      PresPreparada_M430 : Bool;
      PresMultiple_M430 : Bool;
      Bit_07_M430 : Bool;
      RecepOK_M431 : Bool;
      PresNormal_M431 : Bool;
      Ausencia_M431 : Bool;
      PresBloqueo_M431 : Bool;
      Galibo_M431 : Bool;
      PresPreparada_M431 : Bool;
      PresMultiple_M431 : Bool;
      Bit_07_M431 : Bool;
      RecepOK_M432 : Bool;
      PresNormal_M432 : Bool;
      Ausencia_M432 : Bool;
      PresBloqueo_M432 : Bool;
      Galibo_M432 : Bool;
      PresPreparada_M432 : Bool;
      PresMultiple_M432 : Bool;
      Bit_07_M432 : Bool;
      RecepOK_M433 : Bool;
      PresNormal_M433 : Bool;
      Ausencia_M433 : Bool;
      PresBloqueo_M433 : Bool;
      Galibo_M433 : Bool;
      PresPreparada_M433 : Bool;
      PresMultiple_M433 : Bool;
      Bit_07_M433 : Bool;
      RecepOK_M434 : Bool;
      PresNormal_M434 : Bool;
      Ausencia_M434 : Bool;
      PresBloqueo_M434 : Bool;
      Galibo_M434 : Bool;
      PresPreparada_M434 : Bool;
      PresMultiple_M434 : Bool;
      Bit_07_M434 : Bool;
      RecepOK_M435 : Bool;
      PresNormal_M435 : Bool;
      Ausencia_M435 : Bool;
      PresBloqueo_M435 : Bool;
      Galibo_M435 : Bool;
      PresPreparada_M435 : Bool;
      PresMultiple_M435 : Bool;
      Bit_07_M435 : Bool;
      RecepOK_M436 : Bool;
      PresNormal_M436 : Bool;
      Ausencia_M436 : Bool;
      PresBloqueo_M436 : Bool;
      Galibo_M436 : Bool;
      PresPreparada_M436 : Bool;
      PresMultiple_M436 : Bool;
      Bit_07_M436 : Bool;
      RecepOK_M437 : Bool;
      PresNormal_M437 : Bool;
      Ausencia_M437 : Bool;
      PresBloqueo_M437 : Bool;
      Galibo_M437 : Bool;
      PresPreparada_M437 : Bool;
      PresMultiple_M437 : Bool;
      Bit_07_M437 : Bool;
      RecepOK_M438 : Bool;
      PresNormal_M438 : Bool;
      Ausencia_M438 : Bool;
      PresBloqueo_M438 : Bool;
      Galibo_M438 : Bool;
      PresPreparada_M438 : Bool;
      PresMultiple_M438 : Bool;
      Bit_07_M438 : Bool;
      RecepOK_M439 : Bool;
      PresNormal_M439 : Bool;
      Ausencia_M439 : Bool;
      PresBloqueo_M439 : Bool;
      Galibo_M439 : Bool;
      PresPreparada_M439 : Bool;
      PresMultiple_M439 : Bool;
      Bit_07_M439 : Bool;
      RecepOK_M440 : Bool;
      PresNormal_M440 : Bool;
      Ausencia_M440 : Bool;
      PresBloqueo_M440 : Bool;
      Galibo_M440 : Bool;
      PresPreparada_M440 : Bool;
      PresMultiple_M440 : Bool;
      Bit_07_M440 : Bool;
      RecepOK_M441 : Bool;
      PresNormal_M441 : Bool;
      Ausencia_M441 : Bool;
      PresBloqueo_M441 : Bool;
      Galibo_M441 : Bool;
      PresPreparada_M441 : Bool;
      PresMultiple_M441 : Bool;
      Bit_07_M441 : Bool;
      RecepOK_M442 : Bool;
      PresNormal_M442 : Bool;
      Ausencia_M442 : Bool;
      PresBloqueo_M442 : Bool;
      Galibo_M442 : Bool;
      PresPreparada_M442 : Bool;
      PresMultiple_M442 : Bool;
      Bit_07_M442 : Bool;
      RecepOK_M443 : Bool;
      PresNormal_M443 : Bool;
      Ausencia_M443 : Bool;
      PresBloqueo_M443 : Bool;
      Galibo_M443 : Bool;
      PresPreparada_M443 : Bool;
      PresMultiple_M443 : Bool;
      Bit_07_M443 : Bool;
      RecepOK_M444 : Bool;
      PresNormal_M444 : Bool;
      Ausencia_M444 : Bool;
      PresBloqueo_M444 : Bool;
      Galibo_M444 : Bool;
      PresPreparada_M444 : Bool;
      PresMultiple_M444 : Bool;
      Bit_07_M444 : Bool;
      RecepOK_M445 : Bool;
      PresNormal_M445 : Bool;
      Ausencia_M445 : Bool;
      PresBloqueo_M445 : Bool;
      Galibo_M445 : Bool;
      PresPreparada_M445 : Bool;
      PresMultiple_M445 : Bool;
      Bit_07_M445 : Bool;
      RecepOK_M446 : Bool;
      PresNormal_M446 : Bool;
      Ausencia_M446 : Bool;
      PresBloqueo_M446 : Bool;
      Galibo_M446 : Bool;
      PresPreparada_M446 : Bool;
      PresMultiple_M446 : Bool;
      Bit_07_M446 : Bool;
      RecepOK_M447 : Bool;
      PresNormal_M447 : Bool;
      Ausencia_M447 : Bool;
      PresBloqueo_M447 : Bool;
      Galibo_M447 : Bool;
      PresPreparada_M447 : Bool;
      PresMultiple_M447 : Bool;
      Bit_07_M447 : Bool;
      RecepOK_M448 : Bool;
      PresNormal_M448 : Bool;
      Ausencia_M448 : Bool;
      PresBloqueo_M448 : Bool;
      Galibo_M448 : Bool;
      PresPreparada_M448 : Bool;
      PresMultiple_M448 : Bool;
      Bit_07_M448 : Bool;
      RecepOK_M449 : Bool;
      PresNormal_M449 : Bool;
      Ausencia_M449 : Bool;
      PresBloqueo_M449 : Bool;
      Galibo_M449 : Bool;
      PresPreparada_M449 : Bool;
      PresMultiple_M449 : Bool;
      Bit_07_M449 : Bool;
      RecepOK_M450 : Bool;
      PresNormal_M450 : Bool;
      Ausencia_M450 : Bool;
      PresBloqueo_M450 : Bool;
      Galibo_M450 : Bool;
      PresPreparada_M450 : Bool;
      PresMultiple_M450 : Bool;
      Bit_07_M450 : Bool;
      RecepOK_M451 : Bool;
      PresNormal_M451 : Bool;
      Ausencia_M451 : Bool;
      PresBloqueo_M451 : Bool;
      Galibo_M451 : Bool;
      PresPreparada_M451 : Bool;
      PresMultiple_M451 : Bool;
      Bit_07_M451 : Bool;
      RecepOK_M452 : Bool;
      PresNormal_M452 : Bool;
      Ausencia_M452 : Bool;
      PresBloqueo_M452 : Bool;
      Galibo_M452 : Bool;
      PresPreparada_M452 : Bool;
      PresMultiple_M452 : Bool;
      Bit_07_M452 : Bool;
      RecepOK_M453 : Bool;
      PresNormal_M453 : Bool;
      Ausencia_M453 : Bool;
      PresBloqueo_M453 : Bool;
      Galibo_M453 : Bool;
      PresPreparada_M453 : Bool;
      PresMultiple_M453 : Bool;
      Bit_07_M453 : Bool;
      RecepOK_M454 : Bool;
      PresNormal_M454 : Bool;
      Ausencia_M454 : Bool;
      PresBloqueo_M454 : Bool;
      Galibo_M454 : Bool;
      PresPreparada_M454 : Bool;
      PresMultiple_M454 : Bool;
      Bit_07_M454 : Bool;
      RecepOK_M455 : Bool;
      PresNormal_M455 : Bool;
      Ausencia_M455 : Bool;
      PresBloqueo_M455 : Bool;
      Galibo_M455 : Bool;
      PresPreparada_M455 : Bool;
      PresMultiple_M455 : Bool;
      Bit_07_M455 : Bool;
      RecepOK_M456 : Bool;
      PresNormal_M456 : Bool;
      Ausencia_M456 : Bool;
      PresBloqueo_M456 : Bool;
      Galibo_M456 : Bool;
      PresPreparada_M456 : Bool;
      PresMultiple_M456 : Bool;
      Bit_07_M456 : Bool;
      RecepOK_M457 : Bool;
      PresNormal_M457 : Bool;
      Ausencia_M457 : Bool;
      PresBloqueo_M457 : Bool;
      Galibo_M457 : Bool;
      PresPreparada_M457 : Bool;
      PresMultiple_M457 : Bool;
      Bit_07_M457 : Bool;
      RecepOK_M458 : Bool;
      PresNormal_M458 : Bool;
      Ausencia_M458 : Bool;
      PresBloqueo_M458 : Bool;
      Galibo_M458 : Bool;
      PresPreparada_M458 : Bool;
      PresMultiple_M458 : Bool;
      Bit_07_M458 : Bool;
      RecepOK_M459 : Bool;
      PresNormal_M459 : Bool;
      Ausencia_M459 : Bool;
      PresBloqueo_M459 : Bool;
      Galibo_M459 : Bool;
      PresPreparada_M459 : Bool;
      PresMultiple_M459 : Bool;
      Bit_07_M459 : Bool;
      RecepOK_M460 : Bool;
      PresNormal_M460 : Bool;
      Ausencia_M460 : Bool;
      PresBloqueo_M460 : Bool;
      Galibo_M460 : Bool;
      PresPreparada_M460 : Bool;
      PresMultiple_M460 : Bool;
      Bit_07_M460 : Bool;
      RecepOK_M461 : Bool;
      PresNormal_M461 : Bool;
      Ausencia_M461 : Bool;
      PresBloqueo_M461 : Bool;
      Galibo_M461 : Bool;
      PresPreparada_M461 : Bool;
      PresMultiple_M461 : Bool;
      Bit_07_M461 : Bool;
      RecepOK_M462 : Bool;
      PresNormal_M462 : Bool;
      Ausencia_M462 : Bool;
      PresBloqueo_M462 : Bool;
      Galibo_M462 : Bool;
      PresPreparada_M462 : Bool;
      PresMultiple_M462 : Bool;
      Bit_07_M462 : Bool;
      RecepOK_M463 : Bool;
      PresNormal_M463 : Bool;
      Ausencia_M463 : Bool;
      PresBloqueo_M463 : Bool;
      Galibo_M463 : Bool;
      PresPreparada_M463 : Bool;
      PresMultiple_M463 : Bool;
      Bit_07_M463 : Bool;
      RecepOK_M464 : Bool;
      PresNormal_M464 : Bool;
      Ausencia_M464 : Bool;
      PresBloqueo_M464 : Bool;
      Galibo_M464 : Bool;
      PresPreparada_M464 : Bool;
      PresMultiple_M464 : Bool;
      Bit_07_M464 : Bool;
      RecepOK_M465 : Bool;
      PresNormal_M465 : Bool;
      Ausencia_M465 : Bool;
      PresBloqueo_M465 : Bool;
      Galibo_M465 : Bool;
      PresPreparada_M465 : Bool;
      PresMultiple_M465 : Bool;
      Bit_07_M465 : Bool;
      RecepOK_M466 : Bool;
      PresNormal_M466 : Bool;
      Ausencia_M466 : Bool;
      PresBloqueo_M466 : Bool;
      Galibo_M466 : Bool;
      PresPreparada_M466 : Bool;
      PresMultiple_M466 : Bool;
      Bit_07_M466 : Bool;
      RecepOK_M467 : Bool;
      PresNormal_M467 : Bool;
      Ausencia_M467 : Bool;
      PresBloqueo_M467 : Bool;
      Galibo_M467 : Bool;
      PresPreparada_M467 : Bool;
      PresMultiple_M467 : Bool;
      Bit_07_M467 : Bool;
      RecepOK_M468 : Bool;
      PresNormal_M468 : Bool;
      Ausencia_M468 : Bool;
      PresBloqueo_M468 : Bool;
      Galibo_M468 : Bool;
      PresPreparada_M468 : Bool;
      PresMultiple_M468 : Bool;
      Bit_07_M468 : Bool;
      RecepOK_M469 : Bool;
      PresNormal_M469 : Bool;
      Ausencia_M469 : Bool;
      PresBloqueo_M469 : Bool;
      Galibo_M469 : Bool;
      PresPreparada_M469 : Bool;
      PresMultiple_M469 : Bool;
      Bit_07_M469 : Bool;
      RecepOK_M470 : Bool;
      PresNormal_M470 : Bool;
      Ausencia_M470 : Bool;
      PresBloqueo_M470 : Bool;
      Galibo_M470 : Bool;
      PresPreparada_M470 : Bool;
      PresMultiple_M470 : Bool;
      Bit_07_M470 : Bool;
      RecepOK_M471 : Bool;
      PresNormal_M471 : Bool;
      Ausencia_M471 : Bool;
      PresBloqueo_M471 : Bool;
      Galibo_M471 : Bool;
      PresPreparada_M471 : Bool;
      PresMultiple_M471 : Bool;
      Bit_07_M471 : Bool;
      RecepOK_M472 : Bool;
      PresNormal_M472 : Bool;
      Ausencia_M472 : Bool;
      PresBloqueo_M472 : Bool;
      Galibo_M472 : Bool;
      PresPreparada_M472 : Bool;
      PresMultiple_M472 : Bool;
      Bit_07_M472 : Bool;
      RecepOK_M473 : Bool;
      PresNormal_M473 : Bool;
      Ausencia_M473 : Bool;
      PresBloqueo_M473 : Bool;
      Galibo_M473 : Bool;
      PresPreparada_M473 : Bool;
      PresMultiple_M473 : Bool;
      Bit_07_M473 : Bool;
      RecepOK_M474 : Bool;
      PresNormal_M474 : Bool;
      Ausencia_M474 : Bool;
      PresBloqueo_M474 : Bool;
      Galibo_M474 : Bool;
      PresPreparada_M474 : Bool;
      PresMultiple_M474 : Bool;
      Bit_07_M474 : Bool;
      RecepOK_M475 : Bool;
      PresNormal_M475 : Bool;
      Ausencia_M475 : Bool;
      PresBloqueo_M475 : Bool;
      Galibo_M475 : Bool;
      PresPreparada_M475 : Bool;
      PresMultiple_M475 : Bool;
      Bit_07_M475 : Bool;
      RecepOK_M476 : Bool;
      PresNormal_M476 : Bool;
      Ausencia_M476 : Bool;
      PresBloqueo_M476 : Bool;
      Galibo_M476 : Bool;
      PresPreparada_M476 : Bool;
      PresMultiple_M476 : Bool;
      Bit_07_M476 : Bool;
      RecepOK_M477 : Bool;
      PresNormal_M477 : Bool;
      Ausencia_M477 : Bool;
      PresBloqueo_M477 : Bool;
      Galibo_M477 : Bool;
      PresPreparada_M477 : Bool;
      PresMultiple_M477 : Bool;
      Bit_07_M477 : Bool;
      RecepOK_M478 : Bool;
      PresNormal_M478 : Bool;
      Ausencia_M478 : Bool;
      PresBloqueo_M478 : Bool;
      Galibo_M478 : Bool;
      PresPreparada_M478 : Bool;
      PresMultiple_M478 : Bool;
      Bit_07_M478 : Bool;
      RecepOK_M479 : Bool;
      PresNormal_M479 : Bool;
      Ausencia_M479 : Bool;
      PresBloqueo_M479 : Bool;
      Galibo_M479 : Bool;
      PresPreparada_M479 : Bool;
      PresMultiple_M479 : Bool;
      Bit_07_M479 : Bool;
      RecepOK_M480 : Bool;
      PresNormal_M480 : Bool;
      Ausencia_M480 : Bool;
      PresBloqueo_M480 : Bool;
      Galibo_M480 : Bool;
      PresPreparada_M480 : Bool;
      PresMultiple_M480 : Bool;
      Bit_07_M480 : Bool;
      RecepOK_M481 : Bool;
      PresNormal_M481 : Bool;
      Ausencia_M481 : Bool;
      PresBloqueo_M481 : Bool;
      Galibo_M481 : Bool;
      PresPreparada_M481 : Bool;
      PresMultiple_M481 : Bool;
      Bit_07_M481 : Bool;
      RecepOK_M482 : Bool;
      PresNormal_M482 : Bool;
      Ausencia_M482 : Bool;
      PresBloqueo_M482 : Bool;
      Galibo_M482 : Bool;
      PresPreparada_M482 : Bool;
      PresMultiple_M482 : Bool;
      Bit_07_M482 : Bool;
      RecepOK_M483 : Bool;
      PresNormal_M483 : Bool;
      Ausencia_M483 : Bool;
      PresBloqueo_M483 : Bool;
      Galibo_M483 : Bool;
      PresPreparada_M483 : Bool;
      PresMultiple_M483 : Bool;
      Bit_07_M483 : Bool;
      RecepOK_M484 : Bool;
      PresNormal_M484 : Bool;
      Ausencia_M484 : Bool;
      PresBloqueo_M484 : Bool;
      Galibo_M484 : Bool;
      PresPreparada_M484 : Bool;
      PresMultiple_M484 : Bool;
      Bit_07_M484 : Bool;
      RecepOK_M485 : Bool;
      PresNormal_M485 : Bool;
      Ausencia_M485 : Bool;
      PresBloqueo_M485 : Bool;
      Galibo_M485 : Bool;
      PresPreparada_M485 : Bool;
      PresMultiple_M485 : Bool;
      Bit_07_M485 : Bool;
      RecepOK_M486 : Bool;
      PresNormal_M486 : Bool;
      Ausencia_M486 : Bool;
      PresBloqueo_M486 : Bool;
      Galibo_M486 : Bool;
      PresPreparada_M486 : Bool;
      PresMultiple_M486 : Bool;
      Bit_07_M486 : Bool;
      RecepOK_M487 : Bool;
      PresNormal_M487 : Bool;
      Ausencia_M487 : Bool;
      PresBloqueo_M487 : Bool;
      Galibo_M487 : Bool;
      PresPreparada_M487 : Bool;
      PresMultiple_M487 : Bool;
      Bit_07_M487 : Bool;
      RecepOK_M488 : Bool;
      PresNormal_M488 : Bool;
      Ausencia_M488 : Bool;
      PresBloqueo_M488 : Bool;
      Galibo_M488 : Bool;
      PresPreparada_M488 : Bool;
      PresMultiple_M488 : Bool;
      Bit_07_M488 : Bool;
      RecepOK_M489 : Bool;
      PresNormal_M489 : Bool;
      Ausencia_M489 : Bool;
      PresBloqueo_M489 : Bool;
      Galibo_M489 : Bool;
      PresPreparada_M489 : Bool;
      PresMultiple_M489 : Bool;
      Bit_07_M489 : Bool;
      RecepOK_M490 : Bool;
      PresNormal_M490 : Bool;
      Ausencia_M490 : Bool;
      PresBloqueo_M490 : Bool;
      Galibo_M490 : Bool;
      PresPreparada_M490 : Bool;
      PresMultiple_M490 : Bool;
      Bit_07_M490 : Bool;
      RecepOK_M491 : Bool;
      PresNormal_M491 : Bool;
      Ausencia_M491 : Bool;
      PresBloqueo_M491 : Bool;
      Galibo_M491 : Bool;
      PresPreparada_M491 : Bool;
      PresMultiple_M491 : Bool;
      Bit_07_M491 : Bool;
      RecepOK_M492 : Bool;
      PresNormal_M492 : Bool;
      Ausencia_M492 : Bool;
      PresBloqueo_M492 : Bool;
      Galibo_M492 : Bool;
      PresPreparada_M492 : Bool;
      PresMultiple_M492 : Bool;
      Bit_07_M492 : Bool;
      RecepOK_M493 : Bool;
      PresNormal_M493 : Bool;
      Ausencia_M493 : Bool;
      PresBloqueo_M493 : Bool;
      Galibo_M493 : Bool;
      PresPreparada_M493 : Bool;
      PresMultiple_M493 : Bool;
      Bit_07_M493 : Bool;
      RecepOK_M494 : Bool;
      PresNormal_M494 : Bool;
      Ausencia_M494 : Bool;
      PresBloqueo_M494 : Bool;
      Galibo_M494 : Bool;
      PresPreparada_M494 : Bool;
      PresMultiple_M494 : Bool;
      Bit_07_M494 : Bool;
      RecepOK_M495 : Bool;
      PresNormal_M495 : Bool;
      Ausencia_M495 : Bool;
      PresBloqueo_M495 : Bool;
      Galibo_M495 : Bool;
      PresPreparada_M495 : Bool;
      PresMultiple_M495 : Bool;
      Bit_07_M495 : Bool;
      RecepOK_M496 : Bool;
      PresNormal_M496 : Bool;
      Ausencia_M496 : Bool;
      PresBloqueo_M496 : Bool;
      Galibo_M496 : Bool;
      PresPreparada_M496 : Bool;
      PresMultiple_M496 : Bool;
      Bit_07_M496 : Bool;
      RecepOK_M497 : Bool;
      PresNormal_M497 : Bool;
      Ausencia_M497 : Bool;
      PresBloqueo_M497 : Bool;
      Galibo_M497 : Bool;
      PresPreparada_M497 : Bool;
      PresMultiple_M497 : Bool;
      Bit_07_M497 : Bool;
      RecepOK_M498 : Bool;
      PresNormal_M498 : Bool;
      Ausencia_M498 : Bool;
      PresBloqueo_M498 : Bool;
      Galibo_M498 : Bool;
      PresPreparada_M498 : Bool;
      PresMultiple_M498 : Bool;
      Bit_07_M498 : Bool;
      RecepOK_M499 : Bool;
      PresNormal_M499 : Bool;
      Ausencia_M499 : Bool;
      PresBloqueo_M499 : Bool;
      Galibo_M499 : Bool;
      PresPreparada_M499 : Bool;
      PresMultiple_M499 : Bool;
      Bit_07_M499 : Bool;
      RecepOK_M500 : Bool;
      PresNormal_M500 : Bool;
      Ausencia_M500 : Bool;
      PresBloqueo_M500 : Bool;
      Galibo_M500 : Bool;
      PresPreparada_M500 : Bool;
      PresMultiple_M500 : Bool;
      Bit_07_M500 : Bool;
      ByteLIbre_501 : Byte;
      CCPIF : Struct
         Marcha : Bool;
         Paro : Bool;
         Error : Bool;
         Automatico : Bool;
         Remoto : Bool;
         Manual : Bool;
         Bit_06 : Bool;
         Bit_07 : Bool;
         RecepOK : Bool;
         Bit_11 : Bool;
         Bit_12 : Bool;
         Bit_13 : Bool;
         Bit_14 : Bool;
         Bit_15 : Bool;
         Reset_NOK : Bool;
         Reset_OK : Bool;
      END_STRUCT;
      CBOX : Array[1..9] of Struct
         Marcha : Bool;
         Paro : Bool;
         Error : Bool;
         Automatico : Bool;
         Remoto : Bool;
         Manual : Bool;
         Bit_06 : Bool;
         Bit_07 : Bool;
         RecepOK : Bool;
         Bit_11 : Bool;
         Bit_12 : Bool;
         Bit_13 : Bool;
         Bit_14 : Bool;
         Bit_15 : Bool;
         Reset_NOK : Bool;
         Reset_OK : Bool;
      END_STRUCT;
      Codigo_CCPIF : Word;
      Codigo_CBOX : Array[1..9] of Word;
      Especial : Array[1..100] of Word;
   END_VAR
BEGIN
END_DATA_BLOCK
